{attribute addProperty BoxType "EL2212-0000-0020"}
{attribute addProperty Id "StatusAT %I*Status_F0DF9677162"}
{attribute addProperty CRC "3346046110"}
{attribute addProperty SizeInBites "16"}
{attribute addProperty SizeInBytes "2"}
TYPE DOX_Status_Channel_C7709C9E :
STRUCT
	{attribute addProperty Name "Status"}
	Status AT %I* : Status_F0DF9677;
END_STRUCT
END_TYPE

(* stored: Version 1.2.0.0, ProductVersion 3.1.4024.9
   DUT DOX_Status_Channel_C7709C9E: Id {47f6b5c6-89df-4570-a4a0-6746f576e0f4} *)
